FUNCTION_BLOCK RecordEndTime
VAR_INPUT
	EndFlag: BOOL := FALSE;
END_VAR
VAR_OUTPUT
	RecordEndFinish : BOOL :=FALSE;
	EndLo: UDINT;
	EndHi: UDINT;
END_VAR
VAR
	UpTrigDetect: R_TRIG;
	MyTimer: getsystemtime;
END_VAR

//start to get system time
MyTimer();

//detect the trigger: false to true
UpTrigDetect(CLK:=EndFlag);

//record ending Timestamp of initializing period
IF UpTrigDetect.Q THEN
	EndHi := MyTimer.timeHiDW;
	EndLo := MyTimer.timeLoDW;
END_IF
RecordEndFinish :=TRUE;

END_FUNCTION_BLOCK

(* stored: Version 1.1.0.1, ProductVersion 3.1.4024.3
   POU RecordEndTime: Id {fb7fceb2-a488-4893-be5f-8ca7f57f250e}, SpecialFunc None *)
